TYPE "Prod_Halted"
VERSION : 0.1
// Block: Prod_Halted
   STRUCT
      Code : Int;
      Message_N : Int;
   END_STRUCT;

END_TYPE
